PROGRAM StartVis
VAR
	NT_StartProcess_0: NT_StartProcess;
	
END_VAR

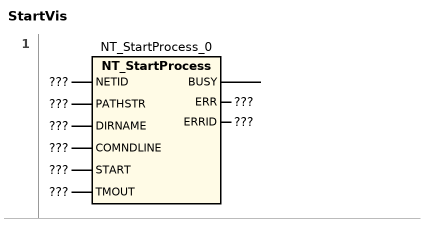
// NETWORK 1
NT_StartProcess_0(); // NT_StartProcess

END_PROGRAM

(* stored: Version 1.1.0.1, ProductVersion 3.1.4024.0
   POU StartVis: Id {d5283a13-9186-4562-8f07-d2d8362f2805}, SpecialFunc None *)
